(* PLC project Tc2_Utilities.stLibVersion_Tc2_Utilities Demo, tc3-libraries-kb TwinCAT 3.1 *)
(* stored: creationDateTime 2026-05-10T11:00:00, modificationDateTime 2026-05-10T11:00:00 *)

PROGRAM P_Demo_stLibVersion_Tc2_Utilities
  VAR
    stMyVer : ST_LibVersion;  (* 本地副本 *)
    bOk : BOOL;  (* 版本检查结果 *)
  END_VAR

            // ============================================================
// Tc2_Utilities.stLibVersion_Tc2_Utilities 演示程序
// ============================================================
// 注意：项目须引用 Tc2_Utilities 与 Tc2_System
// 验证步骤：
//   1. 编译 + 登录
//   2. 在线监视 stMyVer 应显示 2.18.2
//   3. 在线监视 bOk 应为 TRUE
// ============================================================

stMyVer := stLibVersion_Tc2_Utilities;

bOk := F_CmpLibVersion(
    stLibVersion := stLibVersion_Tc2_Utilities,
    iMajor := 2, iMinor := 18, iBuild := 2, iRevision := 0,
    nCmpType := E_CmpLibVersion.GreaterOrEqual
);

          
END_PROGRAM
